Yaskawa INFORM job: SYS-ACK.JBI

/JOB
//NAME SYS-ACK
//POS
///NPOS 0,0,0,0,0,0
//INST
///DATE 2018/07/10 17:56
///ATTR SC,RW,SY
///LVARS 1,0,0,0,0,0,0,0
NOP
*TOP
WAIT IN#(3999)=OFF
DELAY 20
WAIT IN#(3999)=ON
DELAY 20
SET I060 65
*LBL1
DELAY 20
JUMP *LBL1 IF I060<>0
JUMP *TOP
END
